// TIA Portal V18 export
DATA_BLOCK "CTRL_HSC_0_DB_1"   // DB6
// stored: AutoNumber true, InstanceOfName CTRL_HSC, OfSystemLibElement CTRL_HSC, OfSystemLibVersion 1.0
"CTRL_HSC"
   // VAR_INPUT
   //    HSC : HW_HSC;
   //    DIR : Bool;
   //    CV : Bool;
   //    RV : Bool;
   //    PERIOD : Bool;
   //    NEW_DIR : Int;
   //    NEW_CV : DInt;
   //    NEW_RV : DInt;
   //    NEW_PERIOD : Int;
   // END_VAR
   // VAR_OUTPUT
   //    BUSY : Bool;
   //    STATUS : Word;
   // END_VAR
BEGIN
END_DATA_BLOCK
